TYPE ST_PneumaticCylinder :
STRUCT
END_STRUCT
END_TYPE

(* stored: Version 1.1.0.1, ProductVersion 3.1.4026.18
   DUT ST_PneumaticCylinder: Id {a1c89510-1b4f-4861-b699-79fc5925d2e6} *)
